{attribute 'no_explicit_call':= 'do not call this POU directly'}
FUNCTION_BLOCK TValueMonitorEx
VAR
    _Changed : BOOL;
    StoredValue : ARRAY[0..7] OF BYTE;
END_VAR

PROPERTY Changed : BOOL
GET
Changed := _Changed;
END_GET
END_PROPERTY

METHOD Reset
VAR_INPUT
END_VAR
MEMSET(
    destAddr := ADR(StoredValue),
    fillByte  := 16#00,
    n        := SIZEOF(StoredValue));
END_METHOD

METHOD Test : BOOL;
VAR_INPUT
    Value : ANY;
END_VAR
_Changed := 0 <>  MEMCMP(
                    pBuf1 := Value.pValue,
                    pBuf2 := ADR(StoredValue),
                    n     := DINT_TO_UDINT(Value.diSize));
    
IF _Changed THEN
    MEMCPY(
        destAddr := ADR(StoredValue),
        srcAddr  := Value.pValue,
        n        := DINT_TO_UDINT(Value.diSize));
END_IF

Test := _Changed;
END_METHOD

END_FUNCTION_BLOCK

(* stored: Version 1.1.0.1, ProductVersion 3.1.4024.3
   POU TValueMonitorEx: Id {6b5846af-848e-0824-0a24-e0f09726a38e}, SpecialFunc None
   Property Changed: Id {3c3bc936-f576-034a-19b7-f6a5ffc9d4ec}
   Get Get: Id {37c2a605-a4f5-01a7-373c-85bc7a8c26c6}
   Method Reset: Id {57ee03bf-9f21-074c-2e1c-5f316ea5ee90}
   Method Test: Id {ae24e75d-7970-0238-1477-f9aec42558d7} *)
